TYPE ST_RecY : //
STRUCT
	bEnable		                        :BOOL;	
 
	bReady                            :BOOL;  
	bRecOK	 	                   :BOOL;	
	bError				               :BOOL;			
END_STRUCT
END_TYPE

(* stored: Version 1.1.0.1, ProductVersion 3.1.4024.9
   DUT ST_RecY: Id {f88a4ec3-94f0-44c6-9d8d-c4e0b4e91473} *)
